{attribute 'linkalways'} 
{attribute 'no_explicit_call' := 'This FB is a CLASS and must be accessed using methods or properties'}
{attribute 'enable_dynamic_creation'}
FUNCTION_BLOCK FINAL GE_BYTE EXTENDS Node
VAR
	in1 : _BYTE(0);
	in2 : _BYTE(0);
	out : _BOOL(FALSE);
END_VAR

METHOD PUBLIC Clone : I_Node
VAR
	pNode : POINTER TO GE_BYTE;
END_VAR
pNode := __NEW(GE_BYTE);
Clone := pNode^;
END_METHOD

METHOD FB_init : BOOL
VAR_INPUT
	bInitRetains : BOOL; // if TRUE, the retain variables are initialized (warm start / cold start)
	bInCopyCode : BOOL;  // if TRUE, the instance afterwards gets moved into the copy code (online change)
END_VAR
AddInput('in1',THIS^.in1);
AddInput('in2',THIS^.in2);
AddOutput('out', THIS^.out);
END_METHOD

METHOD PROTECTED OnExecute
VAR
END_VAR
out.Value := in1.Value >= in2.Value;
END_METHOD

END_FUNCTION_BLOCK

(* stored: Version 1.1.0.1, ProductVersion 3.1.4024.15
   POU GE_BYTE: Id {77fda2e7-69a7-4ba4-8527-8e4230f4aae7}, SpecialFunc None
   Folder Constructor: Id {ee04c9f5-ae6e-44d4-a8a9-2e77b74bc355}
   Method Clone: Id {8e73aee7-f18f-4dab-83f7-a9961703365e}
   Method FB_init: Id {3c2744a4-8105-400d-8549-a1b542152bdd}
   Method OnExecute: Id {921a8000-69ea-428d-8a4b-4fb9401f8604} *)
